Fanuc KAREL source: CAL_TCP.KL

PROGRAM CAL_TCP
----------------------------------------------------
-- Creation date: 2026.04.22
-- Created by: Zhao Mengkang
----------------------------------------------------
-- Version: 2026.04.22 - 1
----------------------------------------------------
-- Function: Calculate the sphere center from 4 points
----------------------------------------------------
-- Last modified: 2026.04.22
-- Last modified by: Zhao Mengkang
----------------------------------------------------
%COMMENT = 'Test'
%ALPHABETIZE
%NOLOCKGROUP
%NOBUSYLAMP
%NOPAUSESHFT
%NOPAUSE = ERROR + COMMAND + TPENABLE
%SYSTEM

CONST
EPS = 0.000001

VAR
pos1   IN CMOS :XYZWPR
pos2   IN CMOS :XYZWPR
pos3   IN CMOS :XYZWPR
pos4   IN CMOS :XYZWPR

tcp    :XYZWPR
tcp1   :XYZWPR
tcp2   :XYZWPR
tcp3   :XYZWPR
tcp4   :XYZWPR
center :XYZWPR

status :INTEGER
sum_x  :REAL
sum_y  :REAL
sum_z  :REAL

ROUTINE CALCSPH(p1:XYZWPR; p2:XYZWPR; p3:XYZWPR; p4:XYZWPR; center:XYZWPR; status:INTEGER)
VAR
A   :ARRAY[3,3] OF REAL
B   :ARRAY[3] OF REAL
X   :ARRAY[3] OF REAL

P   :ARRAY[4] OF XYZWPR
s1  :REAL

i  :INTEGER
j  :INTEGER
k  :INTEGER
max_row :INTEGER

tmp :REAL
tb  :REAL
factor  :REAL

sum :REAL
BEGIN
    P[1] = p1
    P[2] = p2
    P[3] = p3
    P[4] = p4

    status = 0

    -- Build the linear system from the sphere equations
    -- A * X = B, where X = [cx, cy, cz]
    s1 = p1.x*p1.x + p1.y*p1.y + p1.z*p1.z

    FOR i = 1 TO 3 DO
        j = i + 1
        A[i,1] = 2.0 * (P[j].x - P[1].x)
        A[i,2] = 2.0 * (P[j].y - P[1].y)
        A[i,3] = 2.0 * (P[j].z - P[1].z)

        B[i] = P[j].x*P[j].x + P[j].y*P[j].y + P[j].z*P[j].z - s1
    ENDFOR

    -- Gaussian elimination with partial pivoting
    FOR i = 1 TO 3 DO
        max_row = i

        -- Select the row with the largest pivot element
        FOR k = i + 1 TO 3 DO
            IF ABS(A[k,i]) > ABS(A[max_row,i]) THEN
                max_row = k
            ENDIF
        ENDFOR

        -- Abort if the system is singular or nearly singular
        IF ABS(A[max_row,i]) < EPS THEN
            status = -1
            RETURN
        ENDIF

        -- Swap pivot row into current position
        IF max_row <> i THEN
            FOR k = i TO 3 DO
                tmp = A[i,k]
                A[i,k] = A[max_row,k]
                A[max_row,k] = tmp
            ENDFOR

            tb = B[i]
            B[i] = B[max_row]
            B[max_row] = tb
        ENDIF

        -- Eliminate lower rows
        FOR k = i + 1 TO 3 DO
            factor = A[k,i] / A[i,i]
            FOR j = i TO 3 DO
                A[k,j] = A[k,j] - factor * A[i,j]
            ENDFOR
            B[k] = B[k] - factor * B[i]
        ENDFOR
    ENDFOR

    -- Back substitution to solve X
    FOR i = 3 DOWNTO 1 DO
        sum = B[i]
        FOR j = i + 1 TO 3 DO
            sum = sum - A[i,j] * X[j]
        ENDFOR
        X[i] = sum / A[i,i]
    ENDFOR

    -- Output sphere center
    center.x = X[1]
    center.y = X[2]
    center.z = X[3]
END CALCSPH

ROUTINE WRPR_TO_TCP(p:XYZWPR; center:XYZWPR; tcp:XYZWPR; status:INTEGER)
VAR
rz :REAL
ry :REAL
rx :REAL
c1 :REAL
s1 :REAL
c2 :REAL
s2 :REAL
c3 :REAL
s3 :REAL

T   :ARRAY[4,4] OF REAL
Ti  :ARRAY[4,4] OF REAL

i   :INTEGER
j   :INTEGER
BEGIN
    status = 0

    -- Extract orientation angles from the robot pose
    rx = p.w
    ry = p.p
    rz = p.r

    -- Precompute trigonometric values
    c1 = COS(rz)
    s1 = SIN(rz)
    c2 = COS(ry)
    s2 = SIN(ry)
    c3 = COS(rx)
    s3 = SIN(rx)

    -- Build homogeneous transformation matrix T
    -- Rotation + translation of pose p
    T[1,1] = c1*c2
    T[1,2] = c1*s2*s3 - s1*c3
    T[1,3] = c1*s2*c3 + s1*s3
    T[1,4] = p.x

    T[2,1] = s1*c2
    T[2,2] = s1*s2*s3 + c1*c3
    T[2,3] = s1*s2*c3 - c1*s3
    T[2,4] = p.y

    T[3,1] = -s2
    T[3,2] = c2*s3
    T[3,3] = c2*c3
    T[3,4] = p.z

    T[4,1] = 0
    T[4,2] = 0
    T[4,3] = 0
    T[4,4] = 1

    -- Inverse transform: for rotation matrix, inverse rotation = transpose
    -- Translation part is computed accordingly
    Ti[1,1] = T[1,1]
    Ti[1,2] = T[2,1]
    Ti[1,3] = T[3,1]
    Ti[1,4] = -(Ti[1,1]*T[1,4] + Ti[1,2]*T[2,4] + Ti[1,3]*T[3,4])

    Ti[2,1] = T[1,2]
    Ti[2,2] = T[2,2]
    Ti[2,3] = T[3,2]
    Ti[2,4] = -(Ti[2,1]*T[1,4] + Ti[2,2]*T[2,4] + Ti[2,3]*T[3,4])

    Ti[3,1] = T[1,3]
    Ti[3,2] = T[2,3]
    Ti[3,3] = T[3,3]
    Ti[3,4] = -(Ti[3,1]*T[1,4] + Ti[3,2]*T[2,4] + Ti[3,3]*T[3,4])

    Ti[4,1] = 0
    Ti[4,2] = 0
    Ti[4,3] = 0
    Ti[4,4] = 1

    -- Transform the sphere center into the local tool frame
    tcp.x = Ti[1,1]*center.x + Ti[1,2]*center.y + Ti[1,3]*center.z + Ti[1,4]
    tcp.y = Ti[2,1]*center.x + Ti[2,2]*center.y + Ti[2,3]*center.z + Ti[2,4]
    tcp.z = Ti[3,1]*center.x + Ti[3,2]*center.y + Ti[3,3]*center.z + Ti[3,4]

    -- Only position offset is needed for TCP calibration
    tcp.w = 0
    tcp.p = 0
    tcp.r = 0
END WRPR_TO_TCP

BEGIN

	-- Test Data
    pos1.x = 1575.684
    pos1.y = 141.017
    pos1.z = 382.686
    pos1.w = 121.914
    pos1.p = 19.003
    pos1.r = -10.620

    pos2.x = 1367.624
    pos2.y = 43.138
    pos2.z = 381.901
    pos2.w = 124.729
    pos2.p = -29.614
    pos2.r = 53.708

    pos3.x = 1640.471
    pos3.y = -99.979
    pos3.z = 381.724
    pos3.w = -119.743
    pos3.p = -4.896
    pos3.r = 54.826

    pos4.x = 1450.203
    pos4.y = -144.657
    pos4.z = 382.703
    pos4.w = -131.367
    pos4.p = -40.852
    pos4.r = 4.601

    -- Step 1: calculate the sphere center from four measured points
    CALCSPH(pos1, pos2, pos3, pos4, center, status)
    IF status <> 0 THEN
        ABORT
    ENDIF

    -- Step 2: calculate TCP from each pose and the sphere center
    WRPR_TO_TCP(pos1, center, tcp1, status)
    IF status <> 0 THEN
        ABORT
    ENDIF

    WRPR_TO_TCP(pos2, center, tcp2, status)
    IF status <> 0 THEN
        ABORT
    ENDIF

    WRPR_TO_TCP(pos3, center, tcp3, status)
    IF status <> 0 THEN
        ABORT
    ENDIF

    WRPR_TO_TCP(pos4, center, tcp4, status)
    IF status <> 0 THEN
        ABORT
    ENDIF

    sum_x = (tcp1.x + tcp2.x + tcp3.x + tcp4.x) / 4.0
    sum_y = (tcp1.y + tcp2.y + tcp3.y + tcp4.y) / 4.0
    sum_z = (tcp1.z + tcp2.z + tcp3.z + tcp4.z) / 4.0

    tcp.x = sum_x
    tcp.y = sum_y
    tcp.z = sum_z
    tcp.w = 0
    tcp.p = 0
    tcp.r = 0


END CAL_TCP
